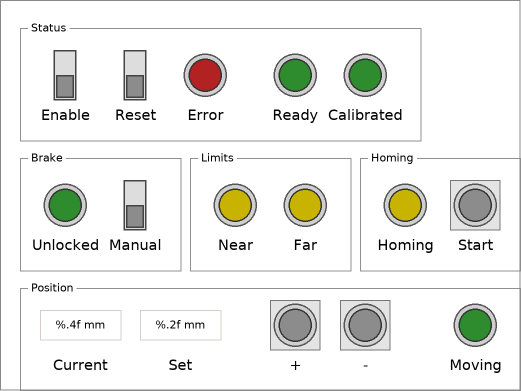
VISUALIZATION Focus  // 521x391
    GroupBox (20,20 401x121), "Status"
        DipSwitch (20,30 50x50), variable: MAIN.FocusControl.enable, behaviour: TOGGLE, style: Switch-DipSwitch-Gray
        DipSwitch (90,30 50x50), variable: MAIN.FocusControl.reset, behaviour: TOGGLE, style: Switch-DipSwitch-Gray
        Label (0,80 91x30), "Enable"
        Label (80,80 71x30), "Reset"
        Lamp1 (160,30 50x50), variable: MAIN.FocusControl.error, style: Lamp-Lamp1-Red
        Label (160,80 51x30), "Error"
        Lamp1 (250,30 50x50), variable: MAIN.FocusControl.ready, style: Lamp-Lamp1-Green
        Lamp1 (320,30 50x50), variable: MAIN.FocusControl.Calibrated, style: Lamp-Lamp1-Green
    Label (270,100 51x30), "Ready"
    Label (330,100 71x30), "Calibrated"
    GroupBox (20,150 161x121), "Brake"
        DipSwitch (90,30 50x50), variable: MAIN.FocusControl.manualUnlock, behaviour: TOGGLE, style: Switch-DipSwitch-Gray
        Label (70,80 91x30), "Manual"
        Lamp1 (20,30 50x50), variable: MAIN.FocusControl.focusUnlocked, style: Lamp-Lamp1-Green
        Label (10,80 71x30), "Unlocked"
    GroupBox (190,150 161x121), "Limits"
        Lamp1 (20,30 50x50), variable: MAIN.FocusControl.inLimitNear, style: Lamp-Lamp1-Yellow
        Label (10,80 71x30), "Near"
        Lamp1 (90,30 50x50), variable: MAIN.FocusControl.inLimitFar, style: Lamp-Lamp1-Yellow
        Label (80,80 71x30), "Far"
    GroupBox (20,280 501x111), "Position"
        Label (20,70 81x30), "Current"
        Label (310,70 71x30), "-"
        Lamp1 (430,20 50x50), variable: MAIN.FocusControl.MoveAxis, style: Lamp-Lamp1-Green
        Label (420,70 71x30), "Moving"
        Textfield (20,30 81x30), "%.4f mm", text variable: MAIN.FocusControl.actualPosition
        Label (120,70 81x30), "Set"
        Textfield (120,30 81x30), "%.2f mm", text variable: MAIN.FocusControl.position
            OnMouseClick: write the text variable via InputWithLimits, min 0, max 100
        PushSwitch (250,20 50x50), variable: MAIN.FocusControl.inward, behaviour: TAP, style: Switch-PushSwitch-Gray
        Label (240,70 71x30), "+"
        PushSwitch (320,20 50x50), variable: MAIN.FocusControl.outward, behaviour: TAP, style: Switch-PushSwitch-Gray
    GroupBox (360,150 161x121), "Homing"
        Lamp1 (20,30 50x50), variable: MAIN.FocusControl.HomeAxis, style: Lamp-Lamp1-Yellow
        Label (10,80 71x30), "Homing"
        Label (80,80 71x30), "Start"
        PushSwitch (90,30 50x50), variable: MAIN.FocusControl.HomeAxis, behaviour: TOGGLE, style: Switch-PushSwitch-Gray
END_VISUALIZATION

(* stored: Version 1.1.0.1, ProductVersion 3.1.4026.8
   Visu Focus: Id {eb878600-4b56-486c-98d0-625f0d713d4b} *)
